(* IEC 61131-3 sources: Industry-PLC-LLM/data/PLCBEAD_repo/PLCBEAD_PLCEmbed-main/PLC-BEAD/Source/GEB/FF_JKE, 1 file *)

(* ---- FF_JKE.ST ---- *)
FUNCTION_BLOCK FF_JKE
	VAR_INPUT
		SET :	BOOL;
		J :	BOOL;
		CLK :	BOOL;
		K :	BOOL;
		RST :	BOOL;
	END_VAR

	VAR_OUTPUT
		Q :	BOOL;
	END_VAR

	VAR
		edge :	BOOL;
	END_VAR

	IF RST OR SET THEN
		Q := NOT RST;
	ELSIF CLK AND NOT edge THEN
		IF J XOR K THEN Q := J;
		ELSE Q := K XOR Q;
		END_IF;
	END_IF;
	edge := CLK;

END_FUNCTION_BLOCK

PROGRAM program0
  VAR
		SET :	BOOL;
		J   :	BOOL;
		CLK :	BOOL;
		K   :	BOOL;
		RST :	BOOL;

		Q :	BOOL;

	func_block : FF_JKE;
  END_VAR
	func_block.SET :=SET;
	func_block.J   :=J  ;
	func_block.CLK :=CLK;
	func_block.K   :=K  ;
	func_block.RST :=RST;
	func_block();
	Q := func_block.Q;
END_PROGRAM
